Staubli VAL3: goTo.pgx

public program goTo(tool x_tTool, mdesc x_mDesc, num x_nMoveType, bool& x_bUnreached[], num x_nIndex)
begin
  // step by step motion
end
